// TIA Portal V17 export
// export: Created 2024-08-26T21:10:49.744185Z, ExportSetting WithDefaults, DisplayName Totally Integrated Automation Portal, DisplayVersion V17 Update 7, DisplayName TIA Portal Openness, DisplayVersion V17 Update 7, DisplayName TIA Portal Version Control Interface, DisplayVersion V17, DisplayName SINAMICS Startdrive Advanced, DisplayVersion V17 SP2, DisplayName SINAMICS Startdrive G110M, G120, G120C, G120D, G120P, G115D, DisplayVersion V17 SP2, DisplayName SINAMICS Startdrive G130, G150, S120, S150, SINAMICS MV, S210, DisplayVersion V17 SP2, DisplayName STEP 7 Professional, DisplayVersion V17 Update 7, DisplayName STEP 7 Safety, DisplayVersion V17 Update 6, DisplayName WinCC Advanced / Unified PC, DisplayVersion V17 Update 7
DATA_BLOCK "LABELS"   // DB6
{ S7_Optimized_Access := 'TRUE' }
VERSION : 0.1
// stored: AutoNumber false, DBAccessibleFromOPCUA true, DBAccessibleFromWebserver true, IsOnlyStoredInLoadMemory false, IsRetainMemResEnabled false, IsWriteProtectedInAS false, MemoryReserve 100
   VAR
      "Previous code" : String := '[) 06 Y40.02.07.01.L P8127005 12V812785841 T9T22202A2B4C1004';
      "Result comp 3" : Int := 0;
      "Result comp 2" : Int := 0;
      "Result comp 1" : Int := 0;
      "Label comp 3" : String := '';
      "Label comp 2" : String := '';
      "Label comp 1" : String := '15';
   END_VAR
   VAR RETAIN
      "Label 1" : Array[0..16] of String[5];   // Label 1
      "Label 2" { ExternalVisible := 'False'} : Array[0..16] of String[5];
      "Label 3" : Array[0..16] of String[5];
      "Label 4" : Array[0..16] of String[5];
      "Label 5" : Array[0..16] of String[5];
      "Label Pos 1" : Array[0..16] of Int;   // label position 1
      "Label Pos 2" : Array[0..16] of Int;
      "Label Pos 3" : Array[0..16] of Int;
      "Label Pos 4" : Array[0..16] of Int;
      "Label Pos 5" : Array[0..16] of Int;   // label position 2
      "Label int" : Array[0..16] of Int;
      Text : Array[0..16] of String[10];   // label text hmi
   END_VAR
   VAR
      Done : Bool := FALSE;
      "Port error" : Bool := FALSE;
      "Port status" : Word := 16#7000;
      "Reset status" : Word := 16#7000;
   END_VAR
   VAR RETAIN
      "Reset done" : Bool := FALSE;
      scanner1 : Bool := TRUE;
      scanner2 : Bool := TRUE;
      scanner3 : Bool := TRUE;
      scanner4 : Bool := FALSE;
      scanner5 : Bool := FALSE;
      scanner6 : Bool := FALSE;
   END_VAR
   VAR
      scannerOn : Bool := TRUE;
      "scann code" : Array[0..1] of String[30];
      "Recive code 2" : String[80] := '';
      labelPrint : String[20] := 'CR24032821X05357';
      NFP : String[35] := '';
      "Recive code" : String[80] := '';
      NDR : Bool := FALSE;
      Error : Bool := FALSE;
      Status : Word := 16#7002;
      Length : UInt := 0;
      labelBlock : Array[0..6] of Bool;
      "Reading scann 1" : String[180] := '';
      "Reading scann 2" : String[180] := 'V008345Y4259698XR011464240801';
      "Extract 5" : Array[0..16] of String[10];
      "Extract 4" : Array[0..16] of String[10];
      "Extract 3" : Array[0..16] of String[10];
      "Extract 2" : Array[0..16] of String[10];
      "Extract 1" : Array[0..16] of String[10];
      "Scanner reading" : Array[0..254] of Char;
      "Previous code scann" : String[40] := '';
      scannerOK2 : Bool := FALSE;
      scannerOK3 : Bool := FALSE;
      scannerOK4 : Bool := FALSE;
      scannerOK5 : Bool := FALSE;
      ScannerOK1 : Bool := FALSE;
      "Scanner length 5" : Array[0..16] of Int;
      "Scanner length 4" : Array[0..16] of Int;
      "Scanner length 3" : Array[0..16] of Int;
      "Scanner length 2" : Array[0..16] of Int;
      "Scanner length 1" : Array[0..16] of Int;
      nestCodeRead : String[80] := '';
      upperCodeRead : String[80] := '';
      angleCodeRead : String[80] := '';
   END_VAR
BEGIN
   "Label 1"[0] := '695';
   "Label 1"[1] := '698';
   "Label 1"[2] := '695';
   "Label 1"[3] := '721';
   "Label 1"[4] := '8721X';
   "Label 1"[5..6] := '698';
   "Label 1"[7..16] := '';
   "Label 2"[0..3] := '06';
   "Label 2"[4] := '1';
   "Label 2"[5] := '06';
   "Label 2"[6] := 'Y4';
   "Label 2"[7..16] := '';
   "Label 3"[0..3] := '06';
   "Label 3"[4] := '';
   "Label 3"[5] := '06';
   "Label 3"[6..16] := '';
   "Label 4"[0..3] := 'Y4';
   "Label 4"[4] := '5/';
   "Label 4"[5] := 'Y4';
   "Label 4"[6] := '5/';
   "Label 4"[7..16] := '';
   "Label 5"[0..6] := '5/';
   "Label 5"[7..16] := '';
   "Label Pos 1"[0..3] := 13;
   "Label Pos 1"[4] := 12;
   "Label Pos 1"[5..6] := 13;
   "Label Pos 1"[7..16] := 0;
   "Label Pos 2"[0..3] := 4;
   "Label Pos 2"[4] := 1;
   "Label Pos 2"[5] := 4;
   "Label Pos 2"[6] := 1;
   "Label Pos 2"[7..16] := 0;
   "Label Pos 3"[0..3] := 4;
   "Label Pos 3"[4] := 0;
   "Label Pos 3"[5] := 4;
   "Label Pos 3"[6..16] := 0;
   "Label Pos 4"[0..3] := 1;
   "Label Pos 4"[4] := 20;
   "Label Pos 4"[5] := 1;
   "Label Pos 4"[6] := 20;
   "Label Pos 4"[7..16] := 0;
   "Label Pos 5"[0..6] := 20;
   "Label Pos 5"[7..16] := 0;
   "Label int"[0] := 151;
   "Label int"[1..16] := 0;
   Text[0] := '';
   Text[1] := 'NEST';
   Text[2] := 'UPPER1';
   Text[3] := 'ANGLE';
   Text[4] := 'UPPER2';
   Text[5..16] := '';
   "scann code"[0..1] := '';
   labelBlock[0..6] := FALSE;
   "Extract 5"[0..16] := '';
   "Extract 4"[0..16] := '';
   "Extract 3"[0..16] := '';
   "Extract 2"[0..16] := '';
   "Extract 1"[0..16] := '';
   "Scanner reading"[0] := '$L';
   "Scanner reading"[1] := '†';
   "Scanner reading"[2] := '$L';
   "Scanner reading"[3] := '†';
   "Scanner reading"[4] := '$L';
   "Scanner reading"[5] := '†';
   "Scanner reading"[6] := '$00';
   "Scanner reading"[7] := '$1E';
   "Scanner reading"[8] := 'B';
   "Scanner reading"[9..10] := '0';
   "Scanner reading"[11] := '2';
   "Scanner reading"[12] := '3';
   "Scanner reading"[13] := '9';
   "Scanner reading"[14] := '0';
   "Scanner reading"[15] := 'W';
   "Scanner reading"[16] := '4';
   "Scanner reading"[17] := '2';
   "Scanner reading"[18] := '6';
   "Scanner reading"[19] := '8';
   "Scanner reading"[20] := '7';
   "Scanner reading"[21] := '2';
   "Scanner reading"[22] := '1';
   "Scanner reading"[23] := 'X';
   "Scanner reading"[24] := 'R';
   "Scanner reading"[25] := '0';
   "Scanner reading"[26..27] := '1';
   "Scanner reading"[28] := '4';
   "Scanner reading"[29] := '6';
   "Scanner reading"[30] := '4';
   "Scanner reading"[31] := '2';
   "Scanner reading"[32] := '4';
   "Scanner reading"[33] := '0';
   "Scanner reading"[34] := '2';
   "Scanner reading"[35] := '0';
   "Scanner reading"[36] := '1';
   "Scanner reading"[37] := '$R';
   "Scanner reading"[38..135] := '$00';
   "Scanner reading"[136..254] := ' ';
   "Scanner length 5"[0] := 0;
   "Scanner length 5"[1] := 3;
   "Scanner length 5"[2..16] := 0;
   "Scanner length 4"[0] := 0;
   "Scanner length 4"[1] := 3;
   "Scanner length 4"[2..16] := 0;
   "Scanner length 3"[0] := 0;
   "Scanner length 3"[1] := 3;
   "Scanner length 3"[2..16] := 0;
   "Scanner length 2"[0] := 0;
   "Scanner length 2"[1] := 3;
   "Scanner length 2"[2..16] := 0;
   "Scanner length 1"[0] := 5;
   "Scanner length 1"[1] := 3;
   "Scanner length 1"[2..16] := 0;
END_DATA_BLOCK
